FUNCTION_BLOCK Test_TEventHandler_HandlesRaisedEvent EXTENDS TUnitTestbase
VAR_INPUT
END_VAR
VAR_OUTPUT
END_VAR
VAR
    TestEvent : TTestEvent;
    TestEventHandler1 : TTestEventHandler;
    TestEventHandler2 : TTestEventHandler;
    TestEventHandler3 : TTestEventHandler;
    TestEventHandler4 : TTestEventHandler;
    TestEventHandler5 : TTestEventHandler;
END_VAR

TestEvent
    .ClearEventHandlers()
    .AddEventHandler(TestEventHandler1)
    .AddEventHandler(TestEventHandler2)
    .AddEventHandler(TestEventHandler3)
    .AddEventHandler(TestEventHandler4)
    .AddEventHandler(TestEventHandler5);
    
TestEvent.Args.Add_UDINT(21);    
TestEvent.Raise();

Assertion.AssertEquals_BOOL(
    Expected := TRUE,
    Actual   := TestEventHandler1.EventWasRaised,
    VariableName  := 'TestEventHandler1.EventWasRaised');

Assertion.AssertEquals_BOOL(
    Expected := TRUE,
    Actual   := TestEventHandler2.EventWasRaised,
    VariableName  := 'TestEventHandler2.EventWasRaised');

Assertion.AssertEquals_BOOL(
    Expected := TRUE,
    Actual   := TestEventHandler3.EventWasRaised,
    VariableName  := 'TestEventHandler3.EventWasRaised');

Assertion.AssertEquals_BOOL(
    Expected := TRUE,
    Actual   := TestEventHandler4.EventWasRaised,
    VariableName  := 'TestEventHandler4.EventWasRaised');

Assertion.AssertEquals_BOOL(
    Expected := TRUE,
    Actual   := TestEventHandler5.EventWasRaised,
    VariableName  := 'TestEventHandler5.EventWasRaised');

    
Assertion.AssertEquals_UDINT(
    Expected := 21,
    Actual   := TestEventHandler1._EventData,
    VariableName  := 'TestEventHandler1._EventData');
    
Assertion.AssertEquals_UDINT(
    Expected := 21,
    Actual   := TestEventHandler2._EventData,
    VariableName  := 'TestEventHandler2._EventData');
    
Assertion.AssertEquals_UDINT(
    Expected := 21,
    Actual   := TestEventHandler3._EventData,
    VariableName  := 'TestEventHandler3._EventData');
    
Assertion.AssertEquals_UDINT(
    Expected := 21,
    Actual   := TestEventHandler4._EventData,
    VariableName  := 'TestEventHandler4._EventData');
    
Assertion.AssertEquals_UDINT(
    Expected := 21,
    Actual   := TestEventHandler5._EventData,
    VariableName  := 'TestEventHandler5._EventData');
    
TestFinished();

END_FUNCTION_BLOCK

(* stored: Version 1.1.0.1, ProductVersion 3.1.4024.4
   POU Test_TEventHandler_HandlesRaisedEvent: Id {7602da14-53c9-4fd0-a968-0f244eb1dec2}, SpecialFunc None *)
